TYPE E_MeasureMode :
(
	MEAS_MODE_Auto := 0,
	MEAS_MODE_SemiAuto := 1
)USINT;
END_TYPE

(* stored: Version 1.1.0.1, ProductVersion 3.1.0.25
   DUT E_MeasureMode: Id {a3d845dc-35db-425c-95c9-b5e3c47aea90} *)
